INTERFACE I_LinearEncodedDrive EXTENDS I_LinearContinuousDrive, I_EncodedDrive

END_INTERFACE

(* stored: Version 1.1.0.1, ProductVersion 3.1.4024.11
   Itf I_LinearEncodedDrive: Id {f26ff7e7-f36b-4992-82ab-7ca5ddd295cd} *)
